FUNCTION_BLOCK SS3_ifb_ps_Vaccume_Gripper (* Composite FB wrapping other FBs *)
  (* Standard: 61499-2 *)
  (* Version 1.0, 2025-05-16, PS_Transformer_for_Unknown *)
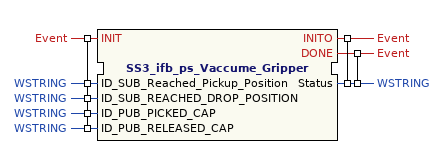
  EVENT_INPUT
    INIT WITH ID_SUB_Reached_Pickup_Position, ID_SUB_REACHED_DROP_POSITION, ID_PUB_PICKED_CAP, ID_PUB_RELEASED_CAP; (* Initialization Request *)
  END_EVENT
  EVENT_OUTPUT
    INITO WITH Status; (* Initialization Confirm *)
    DONE WITH Status; (* Execution Confirmation *)
  END_EVENT
  VAR_INPUT
    ID_SUB_Reached_Pickup_Position : WSTRING;
    ID_SUB_REACHED_DROP_POSITION : WSTRING;
    ID_PUB_PICKED_CAP : WSTRING;
    ID_PUB_RELEASED_CAP : WSTRING;
  END_VAR
  VAR_OUTPUT
    Status : WSTRING; (* Output event qualifier *)
  END_VAR
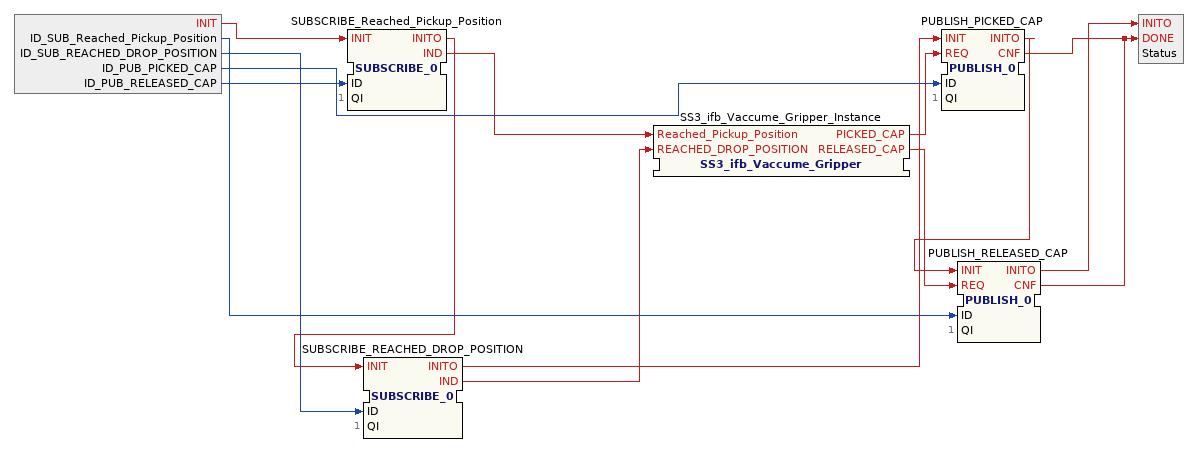
  FBS
    SS3_ifb_Vaccume_Gripper_Instance : SS3_ifb_Vaccume_Gripper;
    SUBSCRIBE_Reached_Pickup_Position : SUBSCRIBE_0(QI := 1);
    SUBSCRIBE_REACHED_DROP_POSITION : SUBSCRIBE_0(QI := 1);
    PUBLISH_PICKED_CAP : PUBLISH_0(QI := 1);
    PUBLISH_RELEASED_CAP : PUBLISH_0(QI := 1);
  END_FBS
  EVENT_CONNECTIONS
    INIT TO SUBSCRIBE_Reached_Pickup_Position.INIT;
    SUBSCRIBE_Reached_Pickup_Position.INITO TO SUBSCRIBE_REACHED_DROP_POSITION.INIT;
    SUBSCRIBE_REACHED_DROP_POSITION.INITO TO PUBLISH_PICKED_CAP.INIT;
    PUBLISH_PICKED_CAP.INITO TO PUBLISH_RELEASED_CAP.INIT;
    PUBLISH_RELEASED_CAP.INITO TO INITO;
    SUBSCRIBE_Reached_Pickup_Position.IND TO SS3_ifb_Vaccume_Gripper_Instance.Reached_Pickup_Position;
    SUBSCRIBE_REACHED_DROP_POSITION.IND TO SS3_ifb_Vaccume_Gripper_Instance.REACHED_DROP_POSITION;
    SS3_ifb_Vaccume_Gripper_Instance.PICKED_CAP TO PUBLISH_PICKED_CAP.REQ;
    SS3_ifb_Vaccume_Gripper_Instance.RELEASED_CAP TO PUBLISH_RELEASED_CAP.REQ;
    PUBLISH_PICKED_CAP.CNF TO DONE;
    PUBLISH_RELEASED_CAP.CNF TO DONE;
  END_CONNECTIONS
  DATA_CONNECTIONS
    ID_SUB_Reached_Pickup_Position TO SUBSCRIBE_Reached_Pickup_Position.ID;
    ID_SUB_REACHED_DROP_POSITION TO SUBSCRIBE_REACHED_DROP_POSITION.ID;
    ID_PUB_PICKED_CAP TO PUBLISH_PICKED_CAP.ID;
    ID_PUB_RELEASED_CAP TO PUBLISH_RELEASED_CAP.ID;
  END_CONNECTIONS
END_FUNCTION_BLOCK
